Yaskawa INFORM job: X2_NOWY2.JBI

/JOB
//NAME X2_NOWY2
//POS
///NPOS 319,319,319,20,0,0
///TOOL 0
///POSTYPE PULSE
///PULSE
C00000=-1579,-114561,-88072,-141,60969,160
C00001=-1579,-126069,-115869,-130,72161,147
C00002=67532,-124352,-115339,-134,72718,152
C00003=81630,-76415,-67707,-7081,99866,75616
C00004=81630,-76414,-67706,-7081,99866,75616
C00005=84756,-88459,-71994,-6618,96608,76878
C00006=84756,-88020,-70779,-6612,96092,76905
C00007=84756,-88291,-71526,-6619,96412,76888
C00008=86383,-83236,-69405,-6430,97828,77376
C00009=86383,-82906,-68386,-6422,97374,77400
C00010=85654,-85197,-69362,-6508,96744,77183
C00011=88190,-77633,-68794,-6246,100461,77872
C00012=91609,-64546,-67425,-5952,106567,78770
C00013=108338,-72557,-69392,-19017,102016,84323
C00014=103994,-87799,-70649,-19047,94316,83966
C00015=101720,-95837,-73131,-19200,91317,83621
C00016=101720,-95093,-71454,-19192,90702,83718
C00017=101720,-95403,-72147,-19196,90955,83679
C00018=102509,-90897,-70406,-19144,92318,83747
C00019=102509,-90529,-69509,-19136,91974,83801
C00020=102070,-93055,-70499,-19166,91217,83763
C00021=103193,-87364,-70534,-19135,94271,83684
C00022=105000,-74500,-64879,-19101,97659,83800
C00023=113069,-60767,-53247,-26239,106025,84622
C00024=112828,-63942,-52646,-27281,108527,83919
C00025=112719,-64865,-51122,-27509,108645,83847
C00026=112853,-61574,-46217,-28469,111221,83243
C00027=112853,-61045,-44714,-28334,110644,83398
C00028=112853,-61574,-46217,-28469,111221,83243
C00029=113196,-56117,-43315,-28575,112240,83113
C00030=113141,-56404,-41984,-28383,111369,83324
C00031=113012,-58464,-43090,-28348,110991,83371
C00032=113141,-56617,-42618,-28443,111618,83258
C00033=126682,-57830,-51235,-23795,116313,87772
C00034=91609,-64546,-67425,-5952,106567,78770
C00035=73590,-134956,-134527,-8565,110042,72105
C00036=73590,-134956,-134527,-8565,110042,72105
C00037=85079,-90579,-82104,-6699,101738,76716
C00038=105233,-99145,-78854,-31145,91869,85162
C00039=90886,-100639,-75930,-30232,80497,82559
C00040=84197,-95229,-69335,-30102,76988,80863
C00041=84197,-94656,-68126,-30150,76597,80967
C00042=84197,-94979,-68806,-30123,76817,80908
C00043=86405,-88952,-66471,-30068,79053,81183
C00044=86405,-88608,-65674,-30094,78780,81256
C00045=85194,-91982,-67001,-30129,77549,81108
C00046=89786,-90500,-68269,-30172,80536,82119
C00047=91499,-86657,-71640,-30020,84676,81700
C00048=78974,-84836,-79700,-7511,102662,74517
C00049=78974,-83060,-72035,-7396,98889,74746
C00050=78731,-83061,-70147,-7399,97713,74732
C00051=78731,-82586,-68642,-7386,97035,74771
C00052=78693,-82844,-69189,-7365,97187,74749
C00053=80468,-78121,-67102,-7173,98481,75288
C00054=80468,-77948,-66494,-7167,98198,75304
C00055=79573,-80363,-67572,-7265,97545,75033
C00056=80252,-78819,-67734,-7202,98493,75213
C00057=80252,-80316,-73749,-7282,101403,75042
C00058=98731,-93358,-79222,-4709,99471,81580
C00059=97921,-96065,-76902,-4782,96613,81409
C00060=97642,-96671,-75645,-4808,95516,81355
C00061=97642,-96038,-74155,-4803,94926,81379
C00062=97642,-96278,-74718,-4805,95148,81370
C00063=99165,-88824,-71799,-4613,97264,81812
C00064=99188,-88439,-71029,-4605,96989,81829
C00065=98601,-91408,-72222,-4678,96166,81658
C00066=99279,-88707,-72907,-4606,98011,81825
C00067=99279,-90964,-80150,-4662,101298,81702
C00068=83031,-73882,-65637,17912,114082,77307
C00069=84799,-81323,-60919,25592,110942,77323
C00070=87066,-81955,-59363,24887,108536,77734
C00071=87066,-80978,-57100,24746,107724,77553
C00072=87066,-81307,-57855,24792,107993,77613
C00073=89010,-75270,-55192,25677,108733,78552
C00074=89357,-73735,-53700,25770,108506,78639
C00075=88474,-76606,-55006,25370,108169,78210
C00076=86155,-69275,-53538,25095,111477,78039
C00077=82305,-66217,-52035,23871,113209,76862
C00078=98731,-93358,-79222,-4709,99471,81580
C00079=87850,-130184,-128808,-6122,98008,77863
C00080=131124,-97291,-82060,-5244,66687,6018
C00081=125790,2337,-22266,-13440,105024,-83634
C00082=119533,36956,22492,-13071,94512,-84678
C00083=111606,23469,-6781,-11265,89839,-86812
C00084=101835,33271,2869,-8999,87620,-9257
C00085=96592,41700,11547,-7901,86106,76285
C00086=96882,40199,11064,-7325,85475,75794
C00087=96412,39571,15762,-7893,82432,76460
C00088=96412,39578,15371,-7890,82674,76445
C00089=96811,43369,19465,-7986,82146,76612
C00090=96811,43369,19923,-7989,81869,76630
C00091=96674,42050,18533,-7957,82032,76574
C00092=96786,43196,17021,-7960,83548,76515
C00093=105692,32729,6227,-9847,85763,79345
C00094=105692,32645,7244,-9851,85104,79396
C00095=105692,32569,8656,-9860,84209,79465
C00096=105692,32584,8289,-9857,84440,79447
C00097=105923,35981,11731,-9908,84100,79551
C00098=105923,35965,12302,-9910,83744,79578
C00099=105845,34812,11128,-9891,83862,79544
C00100=105900,35730,9980,-9889,85029,79471
C00101=105900,36444,4737,-9874,88571,4241
C00102=111606,23469,-6781,-11265,89839,-86812
C00103=109349,27190,646,-10801,86931,-87307
C00104=108816,27234,2830,-10703,85564,-87368
C00105=108816,27153,4539,-10716,84489,-87276
C00106=108816,27166,4149,-10713,84731,-87297
C00107=107956,27551,4528,-10540,84587,-87578
C00108=108965,27264,1619,-10711,86335,-87387
C00109=111260,52324,24435,-15027,98353,-88139
C00110=102462,56667,28820,-9286,105586,-72437
C00111=101371,54153,30717,-9255,103034,-72626
C00112=101300,53253,30624,-9243,102627,-72619
C00113=101300,53374,32279,-9201,101680,-72548
C00114=101300,53356,32072,-9206,101797,-72557
C00115=101042,49940,28251,-9252,102356,-72690
C00116=100773,46580,24617,-9295,102831,-72821
C00117=101300,53356,32072,-9206,101797,-72557
C00118=102175,52590,31226,-9140,102021,-72268
C00119=102630,52208,30804,-9106,102134,-72116
C00120=102175,52590,31226,-9140,102021,-72268
C00121=99428,22928,-9812,-4382,95874,22555
C00122=102095,23568,-1244,-5604,94861,23361
C00123=101997,23184,860,-5428,93239,23419
C00124=101997,23160,1703,-5424,92710,23442
C00125=101997,23183,863,-5429,93237,23419
C00126=102209,25509,3102,-5447,93069,23496
C00127=101997,23183,863,-5429,93237,23419
C00128=101749,19375,-7041,-4715,92641,23427
C00129=101749,19375,-7041,-4715,92641,23427
C00130=102981,33005,7118,-6834,98538,23358
C00131=102660,29046,5283,-6805,97611,23301
C00132=102660,29002,6609,-6789,96777,23347
C00133=102660,29022,5897,-6798,97224,23322
C00134=102541,27735,4980,-6792,97060,7882
C00135=102724,29871,7085,-6794,96879,7954
C00136=102669,29379,3677,-6831,98706,7835
C00137=102669,30744,-3500,-6979,103789,7548
C00138=89085,-61640,-68335,-6227,95184,3424
C00139=129723,10180,-8133,-7222,98462,17027
C00140=105574,29488,-20983,33548,117115,16923
C00141=114766,23108,-3420,30164,101829,15972
C00142=126000,19507,-6631,29272,96237,18805
C00143=125928,21918,3078,29245,93808,18174
C00144=125928,21960,4203,29214,93219,18024
C00145=125927,21943,3808,29209,93425,18075
C00146=125864,24512,6268,29206,93280,18014
C00147=125884,23639,4506,29235,93832,18161
C00148=125884,23787,-988,29454,96866,18937
C00149=117200,23539,-1226,29926,99884,16393
C00150=117161,21121,72,29726,98116,15912
C00151=117144,20144,1246,29621,97051,15628
C00152=117144,20183,2462,29564,96414,15463
C00153=117144,20179,2362,29568,96466,15476
C00154=117212,24135,6125,29546,96194,15431
C00155=117202,23528,1396,29761,98470,16021
C00156=113126,35471,9950,29950,100652,15017
C00157=113126,35383,12410,29782,99292,14657
C00158=113602,35282,14657,29641,97872,14469
C00159=113602,35350,16056,29571,97148,14281
C00160=113602,35312,15354,29605,97509,14375
C00161=114294,35130,15170,29602,97286,14585
C00162=113391,35371,15415,29607,97577,14310
C00163=113626,42883,17073,29878,99977,15031
C00164=136877,41374,10058,-10283,103905,75706
C00165=141001,35831,8537,-10150,102526,77247
C00166=140132,39057,14516,-9459,103035,76976
C00167=140132,39037,16298,-9412,101942,77061
C00168=140132,39036,16078,-9417,102075,77051
C00169=140481,35058,11996,-9419,102579,77132
C00170=140132,39036,16078,-9417,102075,77051
C00171=138905,38111,15122,-9481,102046,76624
C00172=140132,39045,14975,-9447,102749,76998
C00173=140132,39114,13214,-9498,103853,76912
C00174=141320,34178,2051,-14151,101285,76947
C00175=141992,34707,2587,-2039,92766,77188
C00176=132211,33145,3193,16145,89780,75832
C00177=132211,32650,7255,16139,87130,75485
C00178=132167,33411,9664,16155,86089,75333
C00179=132167,33422,9363,16153,86272,75358
C00180=131910,38524,14575,16205,85759,75202
C00181=131910,38519,15135,16208,85424,75158
C00182=131966,37361,13943,16196,85547,75193
C00183=131929,38195,12263,16188,86960,75366
C00184=122451,32022,5983,17773,89556,72453
C00185=122451,31919,7474,17768,88630,72319
C00186=122451,31881,8388,17768,88076,72238
C00187=122451,31892,8078,17768,88262,72265
C00188=122418,36144,12378,17773,87829,72190
C00189=122418,36134,12899,17774,87518,72145
C00190=122425,35123,11870,17773,87626,72164
C00191=122416,36387,11340,17773,88560,72297
C00192=119213,54712,33525,20396,94708,72413
C00193=131575,47506,25138,19197,88561,75788
C00194=127461,43190,24379,29246,85131,74331
C00195=125594,43121,21590,30980,86789,74177
C00196=141320,33353,7524,-13959,97601,77374
C00197=139801,30825,7890,-10211,95473,68752
C00198=139802,30199,7261,-10215,95538,68746
C00199=139884,24100,1063,-10582,96745,77277
C00200=139889,24050,1014,-10582,96750,77278
C00201=131838,40306,17139,3070,104412,75453
C00202=120929,39791,19980,21856,103433,74148
C00203=123594,41501,22617,23894,102676,75270
C00204=120965,41325,24567,29192,101808,74920
C00205=121023,25271,5223,28433,95326,73297
C00206=120372,33506,8504,28624,97501,73589
C00207=120372,33506,8504,28624,97501,7388
C00208=114011,28987,3831,29482,105348,6966
C00209=127254,22780,-708,9297,98542,8796
C00210=130498,22831,169,12202,96699,9956
C00211=128314,21853,36,15870,95950,9465
C00212=117872,21036,1539,32238,96305,7157
C00213=135012,33736,6183,8826,103381,11702
C00214=135092,25600,1604,7767,97772,11260
C00215=129206,23150,2534,20866,94643,10055
C00216=129270,22966,4739,26956,92290,10115
C00217=126431,26011,4689,27524,96578,10067
C00218=115633,44815,18495,18996,108364,-22675
C00219=113931,50187,32287,24759,104059,-23659
C00220=114214,61020,44457,24568,102218,-23946
C00221=113327,59043,39697,24681,104230,-23854
C00222=113549,43239,22387,25049,106471,-23276
C00223=113911,36328,17476,26111,100171,-17352
C00224=113739,31815,13086,26671,97952,-14889
C00225=113784,32033,10394,26825,99526,-14508
C00226=112924,58292,37776,24734,105077,-23825
C00227=109456,25709,2980,23794,97137,-26657
C00228=118237,30699,-4511,-6400,110959,-24971
C00229=106534,-87247,-110627,-560,89262,-27492
C00230=106534,-87247,-110627,-560,89262,-27492
C00231=103790,-60662,-71601,-3492,92371,-24893
C00232=90072,-46297,-51679,-19403,82444,-29914
C00233=88782,-24876,-37241,-19032,94977,-28724
C00234=83056,-19220,-33134,-18691,94035,-30602
C00235=91975,-27497,-33981,-31814,87523,-26891
C00236=93212,-29211,-40642,-31971,90742,-27310
C00237=74629,-7827,-31935,-11254,101997,-33705
C00238=71332,-2618,-22779,-6795,101795,-34320
C00239=78462,-13458,-29551,-16867,94681,-32171
C00240=82147,-18257,-28181,-29567,85461,-30082
C00241=85091,-23046,-35219,-29948,88128,-29642
C00242=83033,-12319,-25680,-29668,87094,-30159
C00243=84406,-14503,-30600,-29861,89239,-30192
C00244=85356,-5858,-28119,-20956,91780,33865
C00245=81588,1895,-16736,-16916,91105,34512
C00246=79661,-5794,-23031,-16691,90641,33907
C00247=79399,-7103,-23567,-16653,90261,33865
C00248=76746,-16078,-29946,-18475,91965,32513
C00249=81974,-12051,-30981,-19262,96095,33689
C00250=98247,-31422,-44950,-19682,96659,36405
C00251=99419,-12339,-27396,-19686,95995,36931
C00252=98336,-20805,-33556,-19612,95212,36674
C00253=97436,-32531,-42916,-18662,91677,32211
C00254=95696,-34091,-42802,-18103,89563,30497
C00255=96230,-30895,-40673,-18159,89998,30622
C00256=92776,-41331,-47434,-14269,83214,21666
C00257=93749,-43799,-52657,-14401,85273,21763
C00258=91043,-39779,-53377,-13904,87247,20611
C00259=86158,-7385,-30463,-15366,102993,69398
C00260=78323,6041,-20316,-6463,111515,89101
C00261=75760,-7515,-27225,-1279,101545,89102
C00262=73720,-14383,-32408,-1291,101175,88413
C00263=73707,-14423,-32438,-1291,101173,88409
C00264=74501,-16417,-33720,-1350,100398,77182
C00265=81364,-12014,-29075,-8477,103574,60369
C00266=76974,-6126,-24441,-8683,103288,58863
C00267=85840,-5383,-30241,-8443,108111,61612
C00268=89409,13061,-14467,-8223,108236,62856
C00269=89565,10966,-11640,-8073,105463,63104
C00270=76842,29074,5202,-8683,103118,58832
C00271=81703,21101,-362,-18048,97571,60243
C00272=83486,19402,-4941,-18704,99513,60525
C00273=85618,-23129,-54211,23,98050,63088
C00274=77730,-75302,-67065,-7588,99691,74263
C00275=69151,-69068,-61329,-2748,102842,72431
C00276=87447,-85862,-67970,5918,101111,78781
C00277=86539,-83533,-63306,15976,104237,78477
C00278=79657,-74315,-62077,14413,109372,76594
C00279=66263,-128090,-130023,6185,104579,72041
C00280=66263,-128090,-130023,6185,104579,72041
C00281=94568,-90015,-76427,6942,102962,81955
C00282=117602,-94880,-71794,18297,96358,89322
C00283=121551,-93080,-69082,18900,94751,90489
C00284=120998,-72436,-50943,33828,103198,79162
C00285=123295,-66551,-41474,44306,102100,75201
C00286=126245,-64319,-39908,46199,101342,75419
C00287=114717,-64735,-41398,43474,107786,72608
C00288=113328,-78138,-63059,20614,107376,72751
C00289=119967,-79989,-67356,-5538,106972,75179
C00290=119601,-81472,-64794,-5557,104619,75157
C00291=101263,-78382,-63761,-10047,103781,68674
C00292=107348,-79714,-62064,-19694,100692,71410
C00293=114949,-81063,-65452,-19014,103658,73736
C00294=107597,-133050,-132520,-1199,109480,70827
C00295=107600,-133050,-132519,-1199,109480,70827
C00296=111097,-94755,-74427,-15472,95771,72593
C00297=108511,-92825,-70401,-15771,93843,71925
C00298=108442,-93231,-70167,-15771,93490,71946
C00299=101417,-63473,-52384,-14930,110878,65868
C00300=99456,-62917,-51924,-15551,110511,65169
C00301=89555,-51250,-43256,-19808,111104,61278
C00302=83325,-44523,-38256,-24472,109539,56579
C00303=85967,-47236,-42901,-22323,110616,58192
C00304=110623,-74300,-66049,-9174,91324,69507
C00305=118006,-113386,-124466,-9637,107827,70792
C00306=118006,-113386,-124466,-9637,107827,70792
C00307=104411,-100441,-71960,-6543,87095,88178
C00308=105456,-99582,-67564,-6467,84927,88642
C00309=110472,-96681,-63053,18266,87626,88449
C00310=100177,-101375,-72775,10447,90542,85701
C00311=127322,-146784,-131564,-384,102103,77635
C00312=127322,-146784,-131564,-384,102103,77635
C00313=128828,-100845,-70585,-1227,88109,75124
C00314=127518,-99136,-66932,-1375,86717,74698
C00315=112854,-98296,-65641,-11209,85327,70513
C00316=128822,-103835,-77575,-9498,91788,75427
C00317=146076,-192209,-136001,-7129,84184,81740
C00318=146076,-192209,-136001,-7129,84184,81740
BC00000=127037,517515,1075193
BC00001=127037,517515,1075193
BC00002=210734,371217,1075193
BC00003=210734,371217,1005131
BC00004=210733,371217,1005128
BC00005=210733,371217,1005125
BC00006=210733,371217,1005125
BC00007=210733,371217,1005125
BC00008=210733,371217,1005125
BC00009=210733,371217,1005125
BC00010=210733,371217,1005125
BC00011=210733,371217,1005125
BC00012=210733,371217,1005125
BC00013=255725,371217,1005125
BC00014=255725,371217,1005125
BC00015=255725,371217,1005125
BC00016=255725,371217,1005125
BC00017=255725,371217,1005125
BC00018=255725,371217,1005125
BC00019=255725,371217,1005125
BC00020=255725,371217,1005125
BC00021=255725,371217,1005125
BC00022=255725,371217,1005125
BC00023=287607,371217,1005125
BC00024=287607,371217,1005125
BC00025=287607,371217,1005125
BC00026=287607,371217,1005125
BC00027=287607,371217,1005125
BC00028=287607,371217,1005125
BC00029=287607,371217,1005125
BC00030=287607,371217,1005125
BC00031=287607,371217,1005125
BC00032=287607,371217,1005125
BC00033=287607,371217,1005125
BC00034=210733,371217,1005125
BC00035=210733,371217,1005125
BC00036=119244,371217,1005125
BC00037=119244,371217,1005125
BC00038=119244,371217,1005125
BC00039=119244,371217,1005125
BC00040=119244,371217,1005125
BC00041=119244,371217,1005125
BC00042=119244,371217,1005125
BC00043=119244,371217,1005125
BC00044=119244,371217,1005125
BC00045=119244,371217,1005125
BC00046=119244,371217,1005125
BC00047=119244,371217,1005125
BC00048=119244,371217,1005121
BC00049=119244,371217,1005121
BC00050=119244,371217,1005121
BC00051=119244,371217,1005121
BC00052=119244,371217,1005121
BC00053=119244,371217,1005121
BC00054=119244,371217,1005121
BC00055=119244,371217,1005121
BC00056=119244,371217,1005121
BC00057=119244,371217,1005121
BC00058=119244,371217,1005121
BC00059=119244,371217,1005121
BC00060=119244,371217,1005121
BC00061=119244,371217,1005121
BC00062=119244,371217,1005121
BC00063=119244,371217,1005121
BC00064=119244,371217,1005121
BC00065=119244,371217,1005121
BC00066=119244,371217,1005121
BC00067=119244,371217,1005121
BC00068=119244,371217,1005121
BC00069=119244,371217,1005121
BC00070=119244,371217,1005121
BC00071=119244,371217,1005121
BC00072=119244,371217,1005121
BC00073=119244,371217,1005121
BC00074=119244,371217,1005121
BC00075=119244,371217,1005121
BC00076=119244,371217,1005121
BC00077=119244,371217,1005121
BC00078=119244,371217,1005121
BC00079=119244,371217,1005121
BC00080=271050,517514,967880
BC00081=271050,517514,967880
BC00082=271050,517514,967880
BC00083=271050,517514,742560
BC00084=271050,517512,742552
BC00085=271050,517512,742552
BC00086=271050,517512,742552
BC00087=271050,517512,742550
BC00088=271050,517512,742550
BC00089=271050,517512,742550
BC00090=271050,517512,742550
BC00091=271050,517512,742550
BC00092=271050,517512,742550
BC00093=271050,517512,742550
BC00094=271050,517512,742550
BC00095=271050,517512,742550
BC00096=271050,517512,742550
BC00097=271050,517512,742550
BC00098=271050,517512,742550
BC00099=271050,517512,742550
BC00100=271050,517512,742550
BC00101=271050,517512,742550
BC00102=271050,517514,742560
BC00103=271050,517513,742557
BC00104=271050,517513,742557
BC00105=271049,517513,742553
BC00106=271049,517513,742553
BC00107=271049,517513,742553
BC00108=271049,517512,742550
BC00109=271049,517512,742550
BC00110=271049,517022,742550
BC00111=271049,517022,742550
BC00112=271049,517022,742550
BC00113=271049,517022,742550
BC00114=271049,517022,742550
BC00115=271049,517022,742550
BC00116=271049,517022,742550
BC00117=271049,517022,742550
BC00118=271049,517022,742550
BC00119=271049,517022,742550
BC00120=271049,517022,742550
BC00121=271049,517024,742547
BC00122=271049,517024,742547
BC00123=271049,517024,742547
BC00124=271049,517024,742547
BC00125=271049,517024,742547
BC00126=271049,517024,742547
BC00127=271049,517024,742547
BC00128=271049,517024,742547
BC00129=291607,517024,742547
BC00130=291607,517024,742547
BC00131=291607,517024,742547
BC00132=291607,517024,742547
BC00133=291607,517024,742547
BC00134=291607,517024,742547
BC00135=291607,517024,742547
BC00136=291607,517024,742547
BC00137=291607,517024,1054319
BC00138=130785,517024,1059413
BC00139=130786,517026,1031640
BC00140=130786,517026,742533
BC00141=130786,517026,742533
BC00142=130786,517026,742533
BC00143=130786,517026,742533
BC00144=130786,517026,742533
BC00145=130786,517026,742530
BC00146=130786,517026,742530
BC00147=130786,517026,742530
BC00148=130786,517026,742530
BC00149=130786,517026,742530
BC00150=130786,517026,742530
BC00151=130786,517026,742530
BC00152=130786,517026,742530
BC00153=130786,517026,742530
BC00154=130786,517026,742530
BC00155=130786,517026,742530
BC00156=130786,517026,742530
BC00157=130786,517026,742530
BC00158=130786,517026,742530
BC00159=130786,517026,742530
BC00160=130786,517026,742530
BC00161=130786,517026,742530
BC00162=130786,517026,742530
BC00163=130786,517026,742530
BC00164=130786,517026,742530
BC00165=130786,517026,742530
BC00166=130786,517026,742530
BC00167=130786,517026,742530
BC00168=130786,517026,742530
BC00169=130786,517026,742530
BC00170=130786,517026,742530
BC00171=130786,517026,742530
BC00172=130786,517026,742530
BC00173=130786,517026,742530
BC00174=130786,517026,742530
BC00175=130786,517026,742530
BC00176=130786,517026,742530
BC00177=130786,517026,742530
BC00178=130786,517026,742530
BC00179=130786,517026,742530
BC00180=130786,517026,742530
BC00181=130786,517026,742530
BC00182=130786,517026,742530
BC00183=130786,517026,742530
BC00184=130786,517026,742530
BC00185=130786,517026,742530
BC00186=130786,517026,742530
BC00187=130786,517026,742530
BC00188=130786,517026,742530
BC00189=130786,517026,742530
BC00190=130786,517026,742530
BC00191=130786,517026,742530
BC00192=130786,517025,742530
BC00193=130786,517026,742527
BC00194=130786,517026,742530
BC00195=130786,517026,742530
BC00196=130786,517026,742530
BC00197=130786,517026,742530
BC00198=130786,517026,742530
BC00199=130786,517026,742530
BC00200=130786,517026,742530
BC00201=130786,517026,742530
BC00202=130786,517026,742530
BC00203=130786,517026,742530
BC00204=130786,517026,742530
BC00205=130786,517026,742530
BC00206=130786,517026,742530
BC00207=130786,517026,742530
BC00208=130786,517026,742530
BC00209=130786,517026,742530
BC00210=130786,517026,742530
BC00211=130786,517026,742530
BC00212=130786,517026,742530
BC00213=130786,517026,742530
BC00214=130786,517026,742530
BC00215=130786,517026,742530
BC00216=130786,517026,742530
BC00217=130786,517026,742530
BC00218=130786,517026,742530
BC00219=130786,517026,742530
BC00220=130786,517026,742530
BC00221=130786,517026,742530
BC00222=130786,517026,742530
BC00223=130786,517026,742530
BC00224=130786,517026,742530
BC00225=130786,517026,742530
BC00226=130786,517026,742530
BC00227=130786,517026,742530
BC00228=130786,517026,742530
BC00229=130786,517026,742530
BC00230=239181,517026,742530
BC00231=239181,441394,742530
BC00232=239181,441394,742530
BC00233=239180,441395,742526
BC00234=239180,441395,742526
BC00235=239180,441395,742526
BC00236=239180,441395,742526
BC00237=239180,441395,742526
BC00238=239180,441395,742526
BC00239=239180,441395,742526
BC00240=239180,441395,742526
BC00241=239180,441395,742526
BC00242=239180,441395,742526
BC00243=239180,441395,742523
BC00244=239180,441395,742523
BC00245=239180,441395,742523
BC00246=239180,441395,742523
BC00247=239180,441395,742523
BC00248=239180,441395,742523
BC00249=239180,441395,742523
BC00250=239180,441395,742523
BC00251=239180,441395,742523
BC00252=239180,441395,742523
BC00253=239180,441395,742523
BC00254=239180,441395,742523
BC00255=239180,441395,742523
BC00256=239180,441395,742523
BC00257=239180,441395,742523
BC00258=239180,441395,742523
BC00259=239180,441395,742523
BC00260=239180,441395,742523
BC00261=239180,441395,742523
BC00262=239180,441395,742523
BC00263=239180,441395,742523
BC00264=239180,441395,742523
BC00265=239180,441395,742523
BC00266=239180,441395,742523
BC00267=239180,441395,742523
BC00268=239180,441395,742523
BC00269=239180,441395,742523
BC00270=239180,441394,742519
BC00271=239180,441394,742519
BC00272=239180,441394,742519
BC00273=239180,441395,742520
BC00274=210733,371217,1005125
BC00275=210733,371217,1005125
BC00276=210734,371218,1005123
BC00277=210734,371218,1005123
BC00278=210734,371218,1005123
BC00279=210734,371218,1005121
BC00280=123056,371218,1005121
BC00281=123056,371218,1005121
BC00282=162204,371218,1005121
BC00283=162204,371218,1005116
BC00284=162204,371218,1005117
BC00285=162204,371218,1005117
BC00286=162204,371218,1005117
BC00287=162204,371218,1005117
BC00288=162204,371218,1005117
BC00289=162204,371218,1005117
BC00290=162204,371218,1005117
BC00291=162204,371218,1005117
BC00292=162204,371218,1005117
BC00293=162204,371218,1005117
BC00294=162204,371218,1005117
BC00295=264253,371217,1005114
BC00296=264253,371217,1005114
BC00297=264253,371217,1005114
BC00298=264253,371217,1005112
BC00299=264253,371217,1005112
BC00300=264253,371217,1005112
BC00301=264250,371217,1005111
BC00302=264252,371217,1005112
BC00303=264253,371217,1005112
BC00304=264253,371217,1005112
BC00305=264253,371217,1005112
BC00306=150415,371217,1056841
BC00307=150415,371217,1056841
BC00308=150415,371217,1056841
BC00309=150415,371217,1056841
BC00310=150415,371217,1056841
BC00311=150415,371217,1056841
BC00312=276067,371217,1056841
BC00313=276067,371217,1056841
BC00314=276067,371217,1056841
BC00315=276067,371217,1056841
BC00316=276067,371217,1056841
BC00317=276067,371217,1056841
BC00318=276067,505629,1056841
EC00000=1527674,-741132
EC00001=1527674,-741132
EC00002=1527674,-741132
EC00003=1527674,-741132
EC00004=1527674,-741132
EC00005=1527674,-741133
EC00006=1527674,-741133
EC00007=1527674,-741133
EC00008=1527674,-741133
EC00009=1527674,-741133
EC00010=1527674,-741133
EC00011=1527674,-741133
EC00012=1527674,-741133
EC00013=1527674,-741133
EC00014=1527674,-741133
EC00015=1527674,-741133
EC00016=1527674,-741133
EC00017=1527674,-741133
EC00018=1527674,-741133
EC00019=1527674,-741133
EC00020=1527674,-741133
EC00021=1527674,-741133
EC00022=1527674,-741133
EC00023=1527674,-741133
EC00024=1527674,-741133
EC00025=1527674,-741133
EC00026=1527674,-741133
EC00027=1527674,-741133
EC00028=1527674,-741133
EC00029=1527674,-741133
EC00030=1527674,-741133
EC00031=1527674,-741133
EC00032=1527674,-741133
EC00033=1527674,-741133
EC00034=1527674,-741133
EC00035=1527674,-741133
EC00036=1527674,-741133
EC00037=1527674,-741133
EC00038=1527674,-741133
EC00039=1527674,-741133
EC00040=1527674,-741133
EC00041=1527674,-741133
EC00042=1527674,-741133
EC00043=1527674,-741133
EC00044=1527674,-741133
EC00045=1527674,-741133
EC00046=1527674,-741133
EC00047=1527674,-741133
EC00048=1527675,-741133
EC00049=1527675,-741133
EC00050=1527675,-741133
EC00051=1527675,-741133
EC00052=1527675,-741133
EC00053=1527675,-741133
EC00054=1527675,-741133
EC00055=1527675,-741133
EC00056=1527675,-741133
EC00057=1527675,-741133
EC00058=1527675,-741133
EC00059=1527675,-741133
EC00060=1527675,-741133
EC00061=1527675,-741133
EC00062=1527675,-741133
EC00063=1527675,-741133
EC00064=1527675,-741133
EC00065=1527675,-741133
EC00066=1527675,-741133
EC00067=1527675,-741133
EC00068=1527675,-741133
EC00069=1527675,-741133
EC00070=1527675,-741133
EC00071=1527675,-741133
EC00072=1527675,-741133
EC00073=1527675,-741133
EC00074=1527675,-741133
EC00075=1527675,-741133
EC00076=1527675,-741133
EC00077=1527675,-741133
EC00078=1527675,-741133
EC00079=1527675,-741133
EC00080=1332361,-741133
EC00081=1332361,-741133
EC00082=1332361,-741133
EC00083=1332361,-741133
EC00084=1332360,-741135
EC00085=1332360,-741135
EC00086=1332360,-741135
EC00087=1332360,-741135
EC00088=1332360,-741135
EC00089=1332360,-741135
EC00090=1332360,-741135
EC00091=1332360,-741135
EC00092=1332360,-741135
EC00093=1332360,-741135
EC00094=1332360,-741135
EC00095=1332360,-741135
EC00096=1332360,-741135
EC00097=1332360,-741135
EC00098=1332360,-741135
EC00099=1332360,-741135
EC00100=1332360,-741135
EC00101=1332360,-741135
EC00102=1332361,-741133
EC00103=1332361,-741134
EC00104=1332361,-741134
EC00105=1332361,-741134
EC00106=1332361,-741134
EC00107=1332361,-741134
EC00108=1332361,-741134
EC00109=1332361,-741134
EC00110=1332361,-741134
EC00111=1332361,-741134
EC00112=1332361,-741134
EC00113=1332361,-741134
EC00114=1332361,-741134
EC00115=1332361,-741134
EC00116=1332361,-741134
EC00117=1332361,-741134
EC00118=1332361,-741134
EC00119=1332361,-741134
EC00120=1332361,-741134
EC00121=1332361,-741134
EC00122=1332361,-741134
EC00123=1332361,-741134
EC00124=1332361,-741134
EC00125=1332361,-741134
EC00126=1332361,-741134
EC00127=1332361,-741134
EC00128=1332361,-741134
EC00129=1332361,-741134
EC00130=1332361,-741134
EC00131=1332361,-741134
EC00132=1332361,-741134
EC00133=1332361,-741134
EC00134=1332361,-741134
EC00135=1332361,-741134
EC00136=1332361,-741134
EC00137=1332361,-741134
EC00138=1332361,-741134
EC00139=1332361,-741135
EC00140=1332361,-741135
EC00141=1332361,-741135
EC00142=1332361,-741135
EC00143=1332361,-741135
EC00144=1332361,-741135
EC00145=1332361,-741135
EC00146=1332361,-741135
EC00147=1332361,-741135
EC00148=1332361,-741135
EC00149=1332361,-741135
EC00150=1332361,-741135
EC00151=1332361,-741135
EC00152=1332361,-741135
EC00153=1332361,-741135
EC00154=1332361,-741135
EC00155=1332361,-741135
EC00156=1332361,-741135
EC00157=1332361,-741135
EC00158=1332361,-741135
EC00159=1332361,-741135
EC00160=1332361,-741135
EC00161=1332361,-741135
EC00162=1332361,-741135
EC00163=1332361,-741135
EC00164=1332361,-741135
EC00165=1332361,-741135
EC00166=1332361,-741135
EC00167=1332361,-741135
EC00168=1332361,-741135
EC00169=1332361,-741135
EC00170=1332361,-741135
EC00171=1332361,-741135
EC00172=1332361,-741135
EC00173=1332361,-741135
EC00174=1332361,-741135
EC00175=1332361,-741135
EC00176=1332361,-741135
EC00177=1332361,-741135
EC00178=1332361,-741135
EC00179=1332361,-741135
EC00180=1332361,-741135
EC00181=1332361,-741135
EC00182=1332361,-741135
EC00183=1332361,-741135
EC00184=1332361,-741135
EC00185=1332361,-741135
EC00186=1332361,-741135
EC00187=1332361,-741135
EC00188=1332361,-741135
EC00189=1332361,-741135
EC00190=1332361,-741135
EC00191=1332361,-741135
EC00192=1332361,-741135
EC00193=1332360,-741134
EC00194=1332361,-741135
EC00195=1332361,-741135
EC00196=1332361,-741135
EC00197=1332361,-741135
EC00198=1332361,-741135
EC00199=1332361,-741135
EC00200=1332361,-741135
EC00201=1332361,-741135
EC00202=1332361,-741135
EC00203=1332361,-741135
EC00204=1332361,-741135
EC00205=1332361,-741135
EC00206=1332361,-741135
EC00207=1332361,-741135
EC00208=1332361,-741135
EC00209=1332361,-741135
EC00210=1332361,-741135
EC00211=1332361,-741135
EC00212=1332361,-741135
EC00213=1332361,-741135
EC00214=1332361,-741135
EC00215=1332361,-741135
EC00216=1332361,-741135
EC00217=1332361,-741135
EC00218=1332361,-741135
EC00219=1332361,-741135
EC00220=1332361,-741135
EC00221=1332361,-741135
EC00222=1332361,-741135
EC00223=1332361,-741135
EC00224=1332361,-741135
EC00225=1332361,-741135
EC00226=1332361,-741135
EC00227=1332361,-741135
EC00228=1332361,-741135
EC00229=1332361,-741135
EC00230=1332361,-741135
EC00231=1332361,-741135
EC00232=1332361,-741135
EC00233=1332361,-741134
EC00234=1332361,-741135
EC00235=1332361,-741135
EC00236=1332361,-741135
EC00237=1332361,-741135
EC00238=1332361,-741135
EC00239=1332361,-741135
EC00240=1332361,-741135
EC00241=1332361,-741135
EC00242=1332361,-741135
EC00243=1332361,-741135
EC00244=1332361,-741135
EC00245=1332361,-741135
EC00246=1332361,-741135
EC00247=1332361,-741135
EC00248=1332361,-741135
EC00249=1332361,-741135
EC00250=1332361,-741135
EC00251=1332361,-741135
EC00252=1332361,-741135
EC00253=1332361,-741135
EC00254=1332361,-741135
EC00255=1332361,-741135
EC00256=1332361,-741135
EC00257=1332361,-741135
EC00258=1332361,-741135
EC00259=1332361,-741135
EC00260=1332361,-741135
EC00261=1332361,-741135
EC00262=1332361,-741135
EC00263=1332361,-741135
EC00264=1332361,-741135
EC00265=1332361,-741135
EC00266=1332361,-741135
EC00267=1332361,-741135
EC00268=1332361,-741135
EC00269=1332361,-741135
EC00270=1332360,-741135
EC00271=1332360,-741135
EC00272=1332360,-741135
EC00273=1332361,-741135
EC00274=1527674,-741133
EC00275=1527674,-741133
EC00276=1527675,-741133
EC00277=1527675,-741133
EC00278=1527675,-741133
EC00279=1527675,-741134
EC00280=1527675,-741134
EC00281=1527675,-741134
EC00282=1527675,-741134
EC00283=1527676,-741134
EC00284=1527676,-741134
EC00285=1527676,-741134
EC00286=1527676,-741134
EC00287=1527676,-741134
EC00288=1527676,-741134
EC00289=1527676,-741134
EC00290=1527676,-741134
EC00291=1527676,-741134
EC00292=1527676,-741134
EC00293=1527676,-741134
EC00294=1527676,-741134
EC00295=1527677,-741134
EC00296=1527677,-741134
EC00297=1527677,-741134
EC00298=1527678,-741134
EC00299=1527678,-741134
EC00300=1527678,-741134
EC00301=1527680,-741134
EC00302=1527679,-741134
EC00303=1527678,-741134
EC00304=1527678,-741134
EC00305=1527678,-741134
EC00306=1527678,-741134
EC00307=1527678,-741134
EC00308=1527678,-741134
EC00309=1527678,-741134
EC00310=1527678,-741134
EC00311=1527678,-741134
EC00312=1527678,-741134
EC00313=1527678,-741134
EC00314=1527678,-741134
EC00315=1527678,-741134
EC00316=1527678,-741134
EC00317=1527678,-741134
EC00318=1527678,-741134
///POSTYPE BASE
///RECTAN
///RCONF 0,0,0,0,1,0,0,0,0,0,0,0,0,0,0,0,0,0,0,0,0,0,0,0
P00006=2.006,1.622,-0.565,0.0000,0.0000,0.0000
P00021=0.073,2.058,-0.109,0.0000,0.0000,0.0000
P00022=2.006,1.622,-0.565,0.0000,0.0000,0.0000
///RCONF 0,0,0,0,0,0,0,0,0,0,0,0,0,0,0,0,0,0,0,0,0,0,0,0
P00023=-2.957,-4.083,2.762,0.0000,0.0000,0.0000
P00024=-1.466,-0.226,-0.419,0.0000,0.0000,0.0000
P00025=3.643,0.007,-2.585,0.0000,0.0000,0.0000
P00026=2.644,0.055,-2.583,0.0000,0.0000,0.0000
P00027=2.278,0.099,-4.210,0.0000,0.0000,0.0000
P00031=-0.170,0.039,-0.647,0.0000,0.0000,0.0000
P00032=-0.423,0.157,3.222,0.0000,0.0000,0.0000
P00033=0.854,-1.099,3.047,0.0000,0.0000,0.0000
///RCONF 0,0,0,0,1,0,0,0,0,0,0,0,0,0,0,0,0,0,0,0,0,0,0,0
P00034=-8.151,9.743,-4.393,0.0000,0.0000,0.0000
///RCONF 0,0,0,0,0,0,0,0,0,0,0,0,0,0,0,0,0,0,0,0,0,0,0,0
P00035=0.390,-0.027,1.040,0.0000,0.0000,0.0000
P00036=-2.434,0.084,0.197,0.0000,0.0000,0.0000
P00037=-1.075,5.090,-3.949,0.0000,0.0000,0.0000
P00038=0.174,-1.527,-10.860,0.0000,0.0000,0.0000
P00050=-0.123,2.174,-1.314,0.0000,0.0000,0.0000
P00051=-5.945,4.696,-10.293,0.0000,0.0000,0.0000
P00052=-0.153,5.586,-7.982,0.0000,0.0000,0.0000
P00053=0.015,-0.644,-4.942,0.0000,0.0000,0.0000
//INST
///DATE 2024/12/19 12:18
///ATTR SC,RW
///GROUP1 RB1,BS1
///GROUP2 ST1
NOP
'PIERWSZA SEKWENCJA
MOVJ C00000 BC00000 VJ=100.00  +MOVJ EC00000 VJ=100.00
MOVJ C00001 BC00001 VJ=100.00  +MOVJ EC00001 VJ=100.00
MOVJ C00002 BC00002 VJ=100.00  +MOVJ EC00002 VJ=100.00
MOVJ C00003 BC00003 VJ=100.00  +MOVJ EC00003 VJ=100.00
SMOVL C00004 BC00004 V=166.7  +MOVJ EC00004
SMOVL C00005 BC00005 V=166.7  +MOVJ EC00005
SREFP 3 C00006 BC00006  +REFP EC00006
CALL JOB:SEARCH-R1-S13D
SET P021 P006
SFTON3D P021
SMOVL C00007 BC00007 V=166.7  +MOVJ EC00007
SMOVL C00008 BC00008 V=166.7  +MOVJ EC00008
SMOVL C00009 BC00009 V=166.7  +MOVJ EC00009
SREFP 3 C00010 BC00010  +REFP EC00010
CALL JOB:SEARCH-R1-S13D
SET P021 P006
SFTON3D P021
SMOVL C00011 BC00011 V=166.7  +MOVJ EC00011
MOVL C00012 BC00012 V=800.0  +MOVJ EC00012 VJ=100.00
SFTOF3D
SMOVL C00013 BC00013 V=1000.0  +MOVJ EC00013
SMOVL C00014 BC00014 V=166.7  +MOVJ EC00014
SMOVL C00015 BC00015 V=166.7  +MOVJ EC00015
SREFP 3 C00016 BC00016  +REFP EC00016
CALL JOB:SEARCH-R1-S13D
SET P022 P006
SFTON3D P022
SMOVL C00017 BC00017 V=166.7  +MOVJ EC00017
SMOVL C00018 BC00018 V=166.7  +MOVJ EC00018
SMOVL C00019 BC00019 V=166.7  +MOVJ EC00019
SREFP 3 C00020 BC00020  +REFP EC00020
CALL JOB:SEARCH-R1-S13D
SET P022 P006
SFTON3D P022
SMOVL C00021 BC00021 V=166.7  +MOVJ EC00021
MOVL C00022 BC00022 V=800.0  +MOVJ EC00022 VJ=100.00
SFTOF3D
SMOVL C00023 BC00023 V=1000.0  +MOVJ EC00023
SMOVL C00024 BC00024 V=800.0  +MOVJ EC00024
SMOVL C00025 BC00025 V=166.7  +MOVJ EC00025
SMOVL C00026 BC00026 V=166.7  +MOVJ EC00026
SREFP 3 C00027 BC00027  +REFP EC00027
CALL JOB:SEARCH-R1-S13D
SET P023 P006
SFTON3D P023
SMOVL C00028 BC00028 V=166.7  +MOVJ EC00028
SMOVL C00029 BC00029 V=166.7  +MOVJ EC00029
SMOVL C00030 BC00030 V=166.7  +MOVJ EC00030
SREFP 3 C00031 BC00031  +REFP EC00031
CALL JOB:SEARCH-R1-S13D
SET P023 P006
SFTON3D P023
SMOVL C00032 BC00032 V=166.7  +MOVJ EC00032
MOVL C00033 BC00033 V=800.0  +MOVJ EC00033 VJ=100.00
SFTOF3D
SMOVL C00034 BC00034 V=800.0  +MOVJ EC00034
MOVJ C00035 BC00035 VJ=100.00  +MOVJ EC00035 VJ=100.00
SMOVL C00036 BC00036 V=1000.0  +MOVJ EC00036
SMOVL C00037 BC00037 V=1000.0  +MOVJ EC00037
SMOVL C00038 BC00038 V=1000.0  +MOVJ EC00038
SMOVL C00039 BC00039 V=166.7  +MOVJ EC00039
SMOVL C00040 BC00040 V=166.7  +MOVJ EC00040
SREFP 3 C00041 BC00041  +REFP EC00041
CALL JOB:SEARCH-R1-S13D
SET P024 P006
SFTON3D P024
SMOVL C00042 BC00042 V=166.7  +MOVJ EC00042
SMOVL C00043 BC00043 V=166.7  +MOVJ EC00043
SMOVL C00044 BC00044 V=166.7  +MOVJ EC00044
SREFP 3 C00045 BC00045  +REFP EC00045
CALL JOB:SEARCH-R1-S13D
SET P024 P006
SFTON3D P024
SMOVL C00046 BC00046 V=166.7  +MOVJ EC00046
MOVL C00047 BC00047 V=800.0  +MOVJ EC00047 VJ=100.00
SMOVL C00048 BC00048 V=1000.0  +MOVJ EC00048
SMOVL C00049 BC00049 V=166.7  +MOVJ EC00049
SMOVL C00050 BC00050 V=166.7  +MOVJ EC00050
SREFP 3 C00051 BC00051  +REFP EC00051
CALL JOB:SEARCH-R1-S13D
SET P025 P006
SFTON3D P025
SMOVL C00052 BC00052 V=166.7  +MOVJ EC00052
SMOVL C00053 BC00053 V=166.7  +MOVJ EC00053
SMOVL C00054 BC00054 V=166.7  +MOVJ EC00054
SREFP 3 C00055 BC00055  +REFP EC00055
CALL JOB:SEARCH-R1-S13D
SET P025 P006
SFTON3D P025
SMOVL C00056 BC00056 V=166.7  +MOVJ EC00056
MOVL C00057 BC00057 V=800.0  +MOVJ EC00057 VJ=100.00
SFTOF3D
SMOVL C00058 BC00058 V=1000.0  +MOVJ EC00058
SMOVL C00059 BC00059 V=166.7  +MOVJ EC00059
SMOVL C00060 BC00060 V=166.7  +MOVJ EC00060
SREFP 3 C00061 BC00061  +REFP EC00061
CALL JOB:SEARCH-R1-S13D
SET P026 P006
SFTON3D P026
SMOVL C00062 BC00062 V=166.7  +MOVJ EC00062
SMOVL C00063 BC00063 V=166.7  +MOVJ EC00063
SMOVL C00064 BC00064 V=166.7  +MOVJ EC00064
SREFP 3 C00065 BC00065  +REFP EC00065
CALL JOB:SEARCH-R1-S13D
SET P026 P006
SFTON3D P026
SMOVL C00066 BC00066 V=166.7  +MOVJ EC00066
MOVL C00067 BC00067 V=800.0  +MOVJ EC00067 VJ=100.00
SFTOF3D
SMOVL C00068 BC00068 V=1000.0  +MOVJ EC00068
SMOVL C00069 BC00069 V=166.7  +MOVJ EC00069
SMOVL C00070 BC00070 V=166.7  +MOVJ EC00070
SREFP 3 C00071 BC00071  +REFP EC00071
CALL JOB:SEARCH-R1-S13D
SET P027 P006
SFTON3D P027
SMOVL C00072 BC00072 V=166.7  +MOVJ EC00072
SMOVL C00073 BC00073 V=166.7  +MOVJ EC00073
SMOVL C00074 BC00074 V=166.7  +MOVJ EC00074
SREFP 3 C00075 BC00075  +REFP EC00075
CALL JOB:SEARCH-R1-S13D
SET P027 P006
SFTON3D P027
SMOVL C00076 BC00076 V=166.7  +MOVJ EC00076
MOVL C00077 BC00077 V=800.0  +MOVJ EC00077 VJ=100.00
SFTOF3D
SMOVL C00078 BC00078 V=1000.0  +MOVJ EC00078
MOVJ C00079 BC00079 VJ=80.00  +MOVJ EC00079 VJ=80.00
'DRUGA SEKWENCJA
MOVJ C00080 BC00080 VJ=100.00  +MOVJ EC00080 VJ=100.00
MOVJ C00081 BC00081 VJ=100.00  +MOVJ EC00081 VJ=100.00
MOVJ C00082 BC00082 VJ=100.00  +MOVJ EC00082 VJ=100.00
SMOVL C00083 BC00083 V=1000.0  +MOVJ EC00083
SMOVL C00084 BC00084 V=333.3  +MOVJ EC00084
SMOVL C00085 BC00085 V=333.3  +MOVJ EC00085
SMOVL C00086 BC00086 V=333.3  +MOVJ EC00086
SREFP 3 C00087 BC00087  +REFP EC00087
CALL JOB:SEARCH-R1-S13D
SET P050 P006
SFTON3D P050
SMOVL C00088 BC00088 V=166.7  +MOVJ EC00088
SMOVL C00089 BC00089 V=166.7  +MOVJ EC00089
SMOVL C00090 BC00090 V=166.7  +MOVJ EC00090
SREFP 3 C00091 BC00091  +REFP EC00091
CALL JOB:SEARCH-R1-S13D
SET P050 P006
SFTON3D P050
SMOVL C00092 BC00092 V=166.7  +MOVJ EC00092
SMOVL C00093 BC00093 V=333.3  +MOVJ EC00093
SFTOF3D
SMOVL C00094 BC00094 V=333.3  +MOVJ EC00094
SREFP 3 C00095 BC00095  +REFP EC00095
CALL JOB:SEARCH-R1-S13D
SET P051 P006
SFTON3D P051
SMOVL C00096 BC00096 V=166.7  +MOVJ EC00096
SMOVL C00097 BC00097 V=166.7  +MOVJ EC00097
SMOVL C00098 BC00098 V=166.7  +MOVJ EC00098
SREFP 3 C00099 BC00099  +REFP EC00099
CALL JOB:SEARCH-R1-S13D
SET P051 P006
SFTON3D P051
SMOVL C00100 BC00100 V=166.7  +MOVJ EC00100
SMOVL C00101 BC00101 V=333.3  +MOVJ EC00101
SMOVL C00102 BC00102 V=333.3  +MOVJ EC00102
SMOVL C00103 BC00103 V=166.7  +MOVJ EC00103
SMOVL C00104 BC00104 V=166.7  +MOVJ EC00104
SREFP 3 C00105 BC00105  +REFP EC00105
CALL JOB:SEARCH-R1-S13D
SET P031 P006
SFTON3D P031
SMOVL C00106 BC00106 V=166.7  +MOVJ EC00106
SREFP 3 C00107 BC00107  +REFP EC00107
CALL JOB:SEARCH-R1-S13D
SET P031 P006
SFTON3D P031
SMOVL C00108 BC00108 V=166.7  +MOVJ EC00108
MOVL C00109 BC00109 V=800.0  +MOVJ EC00109 VJ=100.00
SMOVL C00110 BC00110 V=1000.0  +MOVJ EC00110
SFTOF3D
SMOVL C00111 BC00111 V=166.7  +MOVJ EC00111
SMOVL C00112 BC00112 V=166.7  +MOVJ EC00112
SREFP 3 C00113 BC00113  +REFP EC00113
CALL JOB:SEARCH-R1-S13D
SET P032 P006
SFTON3D P032
SMOVL C00114 BC00114 V=166.7  +MOVJ EC00114
SMOVL C00115 BC00115 V=166.7  +MOVJ EC00115
SREFP 3 C00116 BC00116  +REFP EC00116
CALL JOB:SEARCH-R1-S13D
SET P032 P006
SFTON3D P032
SMOVL C00117 BC00117 V=166.7  +MOVJ EC00117
SMOVL C00118 BC00118 V=166.7  +MOVJ EC00118
SREFP 3 C00119 BC00119  +REFP EC00119
CALL JOB:SEARCH-R1-S13D
SET P032 P006
SFTON3D P032
SMOVL C00120 BC00120 V=166.7  +MOVJ EC00120
MOVL C00121 BC00121 V=800.0  +MOVJ EC00121 VJ=100.00
SFTOF3D
SMOVL C00122 BC00122 V=166.7  +MOVJ EC00122
SMOVL C00123 BC00123 V=166.7  +MOVJ EC00123
SREFP 3 C00124 BC00124  +REFP EC00124
CALL JOB:SEARCH-R1-S13D
SET P033 P006
SFTON3D P033
SMOVL C00125 BC00125 V=166.7  +MOVJ EC00125
SREFP 3 C00126 BC00126  +REFP EC00126
CALL JOB:SEARCH-R1-S13D
SET P033 P006
SFTON3D P033
SMOVL C00127 BC00127 V=166.7  +MOVJ EC00127
MOVL C00128 BC00128 V=800.0  +MOVJ EC00128 VJ=100.00
SFTOF3D
SMOVL C00129 BC00129 V=800.0  +MOVJ EC00129
SMOVL C00130 BC00130 V=166.7  +MOVJ EC00130
SMOVL C00131 BC00131 V=166.7  +MOVJ EC00131
SREFP 3 C00132 BC00132  +REFP EC00132
CALL JOB:SEARCH-R1-S13D
SET P034 P006
SFTON3D P034
SMOVL C00133 BC00133 V=166.7  +MOVJ EC00133
SMOVL C00134 BC00134 V=166.7  +MOVJ EC00134
SREFP 3 C00135 BC00135  +REFP EC00135
CALL JOB:SEARCH-R1-S13D
SET P034 P006
SFTON3D P034
SMOVL C00136 BC00136 V=166.7  +MOVJ EC00136
SFTOF3D
MOVL C00137 BC00137 V=1000.0  +MOVJ EC00137 VJ=100.00
MOVJ C00138 BC00138 VJ=100.00  +MOVJ EC00138 VJ=100.00
SMOVL C00139 BC00139 V=1000.0  +MOVJ EC00139
SMOVL C00140 BC00140 V=1000.0  +MOVJ EC00140
SMOVL C00141 BC00141 V=1000.0  +MOVJ EC00141
SMOVL C00142 BC00142 V=166.7  +MOVJ EC00142
SMOVL C00143 BC00143 V=166.7  +MOVJ EC00143
SREFP 3 C00144 BC00144  +REFP EC00144
CALL JOB:SEARCH-R1-S13D
SET P035 P006
SFTON3D P035
SMOVL C00145 BC00145 V=166.7  +MOVJ EC00145
SREFP 3 C00146 BC00146  +REFP EC00146
CALL JOB:SEARCH-R1-S13D
SET P035 P006
SFTON3D P035
SMOVL C00147 BC00147 V=166.7  +MOVJ EC00147
MOVL C00148 BC00148 V=500.0  +MOVJ EC00148 VJ=100.00
SFTOF3D
SMOVL C00149 BC00149 V=500.0  +MOVJ EC00149
SMOVL C00150 BC00150 V=166.7  +MOVJ EC00150
SMOVL C00151 BC00151 V=166.7  +MOVJ EC00151
SREFP 3 C00152 BC00152  +REFP EC00152
CALL JOB:SEARCH-R1-S13D
SET P036 P006
SFTON3D P036
SMOVL C00153 BC00153 V=166.7  +MOVJ EC00153
SREFP 3 C00154 BC00154  +REFP EC00154
CALL JOB:SEARCH-R1-S13D
SET P036 P006
SFTON3D P036
SMOVL C00155 BC00155 V=166.7  +MOVJ EC00155
SFTOF3D
MOVL C00156 BC00156 V=800.0  +MOVJ EC00156 VJ=100.00
SMOVL C00157 BC00157 V=166.7  +MOVJ EC00157
SMOVL C00158 BC00158 V=166.7  +MOVJ EC00158
SREFP 3 C00159 BC00159  +REFP EC00159
CALL JOB:SEARCH-R1-S13D
SET P038 P006
SFTON3D P038
SMOVL C00160 BC00160 V=166.7  +MOVJ EC00160
SREFP 3 C00161 BC00161  +REFP EC00161
CALL JOB:SEARCH-R1-S13D
SET P038 P006
SFTON3D P038
SMOVL C00162 BC00162 V=166.7  +MOVJ EC00162
MOVL C00163 BC00163 V=800.0  +MOVJ EC00163 VJ=100.00
SFTOF3D
SMOVL C00164 BC00164 V=1000.0  +MOVJ EC00164
SMOVL C00165 BC00165 V=166.7  +MOVJ EC00165
SMOVL C00166 BC00166 V=166.7  +MOVJ EC00166
SREFP 3 C00167 BC00167  +REFP EC00167
CALL JOB:SEARCH-R1-S13D
SET P037 P006
SFTON3D P037
SMOVL C00168 BC00168 V=166.7  +MOVJ EC00168
SREFP 3 C00169 BC00169  +REFP EC00169
CALL JOB:SEARCH-R1-S13D
SET P037 P006
SFTON3D P037
SMOVL C00170 BC00170 V=166.7  +MOVJ EC00170
SREFP 3 C00171 BC00171  +REFP EC00171
CALL JOB:SEARCH-R1-S13D
SET P037 P006
SMOVL C00172 BC00172 V=166.7  +MOVJ EC00172
MOVL C00173 BC00173 V=800.0  +MOVJ EC00173 VJ=100.00
SFTOF3D
SMOVL C00174 BC00174 V=333.3  +MOVJ EC00174
SMOVL C00175 BC00175 V=333.3  +MOVJ EC00175
SMOVL C00176 BC00176 V=333.3  +MOVJ EC00176
SMOVL C00177 BC00177 V=166.7  +MOVJ EC00177
SREFP 3 C00178 BC00178  +REFP EC00178
CALL JOB:SEARCH-R1-S13D
SET P052 P006
SFTON3D P052
SMOVL C00179 BC00179 V=166.7  +MOVJ EC00179
SMOVL C00180 BC00180 V=166.7  +MOVJ EC00180
SMOVL C00181 BC00181 V=166.7  +MOVJ EC00181
SREFP 3 C00182 BC00182  +REFP EC00182
CALL JOB:SEARCH-R1-S13D
SET P052 P006
SFTON3D P052
SMOVL C00183 BC00183 V=166.7  +MOVJ EC00183
SMOVL C00184 BC00184 V=333.3  +MOVJ EC00184
SMOVL C00185 BC00185 V=166.7  +MOVJ EC00185
SREFP 3 C00186 BC00186  +REFP EC00186
CALL JOB:SEARCH-R1-S13D
SET P053 P006
SFTON3D P053
SMOVL C00187 BC00187 V=166.7  +MOVJ EC00187
SMOVL C00188 BC00188 V=166.7  +MOVJ EC00188
SMOVL C00189 BC00189 V=166.7  +MOVJ EC00189
SREFP 3 C00190 BC00190  +REFP EC00190
CALL JOB:SEARCH-R1-S13D
SET P053 P006
SFTON3D P053
SMOVL C00191 BC00191 V=166.7  +MOVJ EC00191
SMOVL C00192 BC00192 V=166.7 PL=0  +MOVJ EC00192
MACRO1 MJ#(0) ARGF10
ARCON
SFTON3D P052
SMOVL C00193 BC00193 V=10.0  +MOVJ EC00193
SMOVL C00194 BC00194 V=10.0  +MOVJ EC00194
ARCOF
SMOVL C00195 BC00195 V=166.7  +MOVJ EC00195
SMOVL C00196 BC00196 V=800.0  +MOVJ EC00196
MACRO1 MJ#(0) ARGF14
SFTON3D P037
SMOVL C00197 BC00197 V=166.7 PL=0  +MOVJ EC00197
ARCON
SMOVL C00198 BC00198 V=10.0  +MOVJ EC00198
SMOVL C00199 BC00199 V=10.0  +MOVJ EC00199
SMOVC C00200 BC00200 V=10.0  +MOVJ EC00200
SMOVC C00201 BC00201 V=10.0  +MOVJ EC00201
SMOVC C00202 BC00202 V=10.0  +MOVJ EC00202
SMOVL C00203 BC00203 V=10.0  +MOVJ EC00203
SMOVL C00204 BC00204 V=10.0  +MOVJ EC00204
ARCOF
SMOVL C00205 BC00205 V=166.7  +MOVJ EC00205
SFTOF3D
MOVJ C00206 BC00206 VJ=100.00  +MOVJ EC00206 VJ=100.00
MOVJ C00207 BC00207 VJ=100.00  +MOVJ EC00207 VJ=100.00
MOVJ C00208 BC00208 VJ=100.00  +MOVJ EC00208 VJ=100.00
MACRO1 MJ#(0) ARGF10
SFTON3D P035
SMOVL C00209 BC00209 V=166.7  +MOVJ EC00209
ARCON
SMOVL C00210 BC00210 V=6.7  +MOVJ EC00210
MOVL C00211 BC00211 V=6.7  +MOVJ EC00211 VJ=100.00
ARCOF
SMOVL C00212 BC00212 V=166.7  +MOVJ EC00212
SFTOF3D
SMOVL C00213 BC00213 V=166.7  +MOVJ EC00213
SFTON3D P036
SMOVL C00214 BC00214 V=166.7  +MOVJ EC00214
ARCON
SMOVL C00215 BC00215 V=5.8  +MOVJ EC00215
SMOVL C00216 BC00216 V=5.8  +MOVJ EC00216
ARCOF
SMOVL C00217 BC00217 V=166.7  +MOVJ EC00217
SFTOF3D
SMOVL C00218 BC00218 V=166.7  +MOVJ EC00218
SFTON3D P038
SMOVL C00219 BC00219 V=166.7  +MOVJ EC00219
ARCON
SMOVL C00220 BC00220 V=8.3  +MOVJ EC00220
ARCOF
SFTOF3D
MOVL C00221 BC00221 V=166.7  +MOVJ EC00221 VJ=80.00
MOVL C00222 BC00222 V=166.7  +MOVJ EC00222 VJ=80.00
SFTON3D P038
MOVL C00223 BC00223 V=166.7  +MOVJ EC00223 VJ=80.00
ARCON
MOVL C00224 BC00224 V=8.3  +MOVJ EC00224 VJ=80.00
ARCOF
MOVL C00225 BC00225 V=166.7  +MOVJ EC00225 VJ=80.00
SMOVL C00226 BC00226 V=166.7  +MOVJ EC00226
SFTOF3D
SMOVL C00227 BC00227 V=666.7  +MOVJ EC00227
SMOVL C00228 BC00228 V=666.7  +MOVJ EC00228
SMOVL C00229 BC00229 V=1000.0  +MOVJ EC00229
SMOVL C00230 BC00230 V=1000.0  +MOVJ EC00230
SMOVL C00231 BC00231 V=1000.0  +MOVJ EC00231
SMOVL C00232 BC00232 V=1000.0  +MOVJ EC00232
SFTON3D P033
SMOVL C00233 BC00233 V=250.0  +MOVJ EC00233
ARCON
SMOVL C00234 BC00234 V=5.8  +MOVJ EC00234
SMOVL C00235 BC00235 V=5.8  +MOVJ EC00235
ARCOF
SFTOF3D
SMOVL C00236 BC00236 V=166.7  +MOVJ EC00236
SMOVL C00237 BC00237 V=166.7  +MOVJ EC00237
SFTON3D P033
SMOVL C00238 BC00238 V=166.7  +MOVJ EC00238
ARCON
SMOVL C00239 BC00239 V=5.8  +MOVJ EC00239
SMOVL C00240 BC00240 V=5.8  +MOVJ EC00240
ARCOF
SMOVL C00241 BC00241 V=250.0  +MOVJ EC00241
MACRO1 MJ#(0) ARGF6
SMOVL C00242 BC00242 V=250.0  +MOVJ EC00242
ARCON
TIMER T=2.00
ARCOF
MOVJ C00243 BC00243 VJ=100.00  +MOVJ EC00243 VJ=100.00
MOVJ C00244 BC00244 VJ=100.00  +MOVJ EC00244 VJ=100.00
MACRO1 MJ#(0) ARGF9
SMOVL C00245 BC00245 V=250.0  +MOVJ EC00245
ARCON
SMOVL C00246 BC00246 V=7.5  +MOVJ EC00246
ARCOF
SMOVL C00247 BC00247 V=7.5  +MOVJ EC00247
ARCON
SMOVL C00248 BC00248 V=7.5  +MOVJ EC00248
ARCOF
SMOVL C00249 BC00249 V=250.0  +MOVJ EC00249
SMOVL C00250 BC00250 V=250.0  +MOVJ EC00250
SFTON3D P031
SMOVL C00251 BC00251 V=250.0  +MOVJ EC00251
ARCON
SMOVL C00252 BC00252 V=6.7  +MOVJ EC00252
ARCOF
SMOVL C00253 BC00253 V=133.3  +MOVJ EC00253
SMOVL C00254 BC00254 V=133.3  +MOVJ EC00254
COMM ARCON
SMOVL C00255 BC00255 V=8.3  +MOVJ EC00255
SMOVL C00256 BC00256 V=8.3  +MOVJ EC00256
ARCOF
SMOVL C00257 BC00257 V=250.0  +MOVJ EC00257
MOVJ C00258 BC00258 VJ=100.00  +MOVJ EC00258 VJ=100.00
SFTOF3D
MOVJ C00259 BC00259 VJ=100.00  +MOVJ EC00259 VJ=100.00
MOVJ C00260 BC00260 VJ=100.00  +MOVJ EC00260 VJ=100.00
SFTON3D P032
SMOVL C00261 BC00261 V=250.0  +MOVJ EC00261
MACRO1 MJ#(0) ARGF14
ARCON
SMOVL C00262 BC00262 V=10.0  +MOVJ EC00262
SMOVC C00263 BC00263 V=10.0  +MOVJ EC00263
SMOVC C00264 BC00264 V=10.0  +MOVJ EC00264
SMOVC C00265 BC00265 V=10.0  +MOVJ EC00265
SMOVL C00266 BC00266 V=8.3  +MOVJ EC00266
ARCOF
SMOVL C00267 BC00267 V=250.0  +MOVJ EC00267
SFTOF3D
SFTON3D P050
SMOVL C00268 BC00268 V=333.3  +MOVJ EC00268
SMOVL C00269 BC00269 V=166.7 PL=0  +MOVJ EC00269
MACRO1 MJ#(0) ARGF10
ARCON
SFTON3D P051
SMOVL C00270 BC00270 V=10.0  +MOVJ EC00270
SMOVL C00271 BC00271 V=10.0  +MOVJ EC00271
ARCOF
SMOVL C00272 BC00272 V=333.3  +MOVJ EC00272
SFTOF3D
SMOVL C00273 BC00273 V=666.7  +MOVJ EC00273
MOVJ C00274 BC00274 VJ=100.00  +MOVJ EC00274 VJ=100.00
SFTON3D P021
SMOVL C00275 BC00275 V=250.0  +MOVJ EC00275
ARCON
SMOVL C00276 BC00276 V=10.0  +MOVJ EC00276
SMOVL C00277 BC00277 V=10.0  +MOVJ EC00277
ARCOF
SMOVL C00278 BC00278 V=250.0  +MOVJ EC00278
SFTOF3D
SMOVL C00279 BC00279 V=833.3  +MOVJ EC00279
SMOVL C00280 BC00280 V=833.3  +MOVJ EC00280
SMOVL C00281 BC00281 V=833.3  +MOVJ EC00281
SMOVL C00282 BC00282 V=833.3  +MOVJ EC00282
SFTON3D P027
SMOVL C00283 BC00283 V=166.7 PL=0  +MOVJ EC00283
ARCON
SMOVL C00284 BC00284 V=10.0  +MOVJ EC00284
SMOVL C00285 BC00285 V=10.0  +MOVJ EC00285
SMOVL C00286 BC00286 V=10.0  +MOVJ EC00286
ARCOF
SMOVL C00287 BC00287 V=333.3  +MOVJ EC00287
SFTOF3D
SMOVL C00288 BC00288 V=333.3  +MOVJ EC00288
SMOVL C00289 BC00289 V=333.3  +MOVJ EC00289
SFTON3D P025
SMOVL C00290 BC00290 V=250.0  +MOVJ EC00290
ARCON
SFTON3D P024
SMOVL C00291 BC00291 V=10.0  +MOVJ EC00291
SMOVL C00292 BC00292 V=10.0  +MOVJ EC00292
ARCOF
SMOVL C00293 BC00293 V=250.0  +MOVJ EC00293
SMOVL C00294 BC00294 V=833.3  +MOVJ EC00294
SMOVL C00295 BC00295 V=833.3  +MOVJ EC00295
SMOVL C00296 BC00296 V=833.3  +MOVJ EC00296
SMOVL C00297 BC00297 V=333.3  +MOVJ EC00297
SFTON3D P022
SMOVL C00298 BC00298 V=166.7  +MOVJ EC00298
ARCON
SMOVL C00299 BC00299 V=10.0  +MOVJ EC00299
SMOVL C00300 BC00300 V=10.0  +MOVJ EC00300
SFTON3D P023
SMOVL C00301 BC00301 V=10.0  +MOVJ EC00301
SMOVL C00302 BC00302 V=10.0  +MOVJ EC00302
ARCOF
SMOVL C00303 BC00303 V=250.0  +MOVJ EC00303
SFTOF3D
MOVJ C00304 BC00304 VJ=100.00  +MOVJ EC00304 VJ=100.00
MOVJ C00305 BC00305 VJ=100.00  +MOVJ EC00305 VJ=100.00
MOVJ C00306 BC00306 VJ=100.00  +MOVJ EC00306 VJ=100.00
MOVJ C00307 BC00307 VJ=100.00  +MOVJ EC00307 VJ=100.00
'DO SPRAWDZENIA CZY TRAFIA
SFTON3D P025
SMOVL C00308 BC00308 V=250.0  +MOVJ EC00308
ARCON
SFTON3D P026
SMOVL C00309 BC00309 V=10.0  +MOVJ EC00309
ARCOF
SMOVL C00310 BC00310 V=800.0  +MOVJ EC00310
SFTOF3D
MOVJ C00311 BC00311 VJ=100.00  +MOVJ EC00311 VJ=100.00
MOVJ C00312 BC00312 VJ=100.00  +MOVJ EC00312 VJ=100.00
MOVJ C00313 BC00313 VJ=100.00  +MOVJ EC00313 VJ=100.00
SFTON3D P021
SMOVL C00314 BC00314 V=800.0  +MOVJ EC00314
ARCON
SFTON3D P022
SMOVL C00315 BC00315 V=10.0  +MOVJ EC00315
ARCOF
SFTOF3D
SMOVL C00316 BC00316 V=250.0  +MOVJ EC00316
SMOVL C00317 BC00317 V=833.3  +MOVJ EC00317
SMOVL C00318 BC00318 V=833.3  +MOVJ EC00318
END
